TYPE Interval :
STRUCT
	startPos : REAL;
	endPos : REAL;
END_STRUCT
END_TYPE

(* stored: Version 1.1.0.1, ProductVersion 3.1.4024.11
   DUT Interval: Id {c6160f0d-4eaf-4650-ba9d-f76549969dfb} *)
